FUNCTION_BLOCK TFallingEdge
VAR
    F_TRIG1 : F_TRIG;
END_VAR

PROPERTY EdgeDetected : BOOL
GET
EdgeDetected := F_TRIG1.Q;
END_GET
END_PROPERTY

METHOD Test : BOOL
VAR_INPUT
    Value : BOOL;
END_VAR
F_TRIG1(CLK := Value);
Test := F_TRIG1.Q;
END_METHOD

END_FUNCTION_BLOCK

(* stored: Version 1.1.0.1, ProductVersion 3.1.4024.3
   POU TFallingEdge: Id {7f65097c-c9a6-0e52-16b8-f5810374ec4f}, SpecialFunc None
   Property EdgeDetected: Id {ff4c5ace-12dc-082b-2194-4cd82b3d41c0}
   Get Get: Id {c79d7714-f2fc-07e5-33d5-8faa3481029f}
   Method Test: Id {1b32f6a7-da3a-081c-2e3a-ba133294f107} *)
